Staubli VAL3: onRun.pgx

public program onRun(string& x_sItem[])
begin
end
